// TIA Portal V15.1 export
// export: Created 2022-12-20T09:13:23.2931876Z, ExportSetting None, DisplayName Totally Integrated Automation Portal, DisplayVersion V15.1 Update 1, DisplayName TIA Portal Openness, DisplayVersion V15.1, DisplayName SINAMICS Startdrive Advanced, DisplayVersion V15.1, DisplayName G130, G150, S120, S150, SINAMICS MV, S210, DisplayVersion V15.1, DisplayName G110M, G120, G120C, G120D, G120P, DisplayVersion V15.1, DisplayName STEP 7 Professional, DisplayVersion V15.1 Update 1, DisplayName STEP 7 Safety, DisplayVersion V15.1, DisplayName WinCC Professional, DisplayVersion V15.1 Update 1, DisplayName SIMATIC Visualization Architect, DisplayVersion V15.1
FUNCTION_BLOCK "SA01_ESTOP_FB"   // FB901, FBD
TITLE = SA01_Estop_FB
{ S7_Optimized_Access := 'TRUE' }
// The block is used to control the estops that are located on SA01
// stored: AutoNumber false, MemoryReserve 100, SetENOAutomatically False
   VAR
      "xxx-xxxx" : "CM_Estop_FB";   // Emergency stop HMI load area xxxx
   END_VAR
BEGIN

REGION Network 1: Call emergency stop HMI load area Stxxx
   // E-stop xxxx
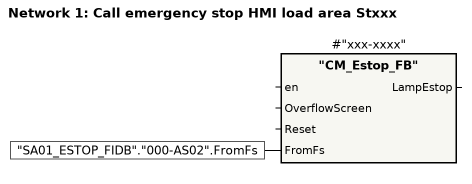
   #"xxx-xxxx"(FromFs := "SA01_ESTOP_FIDB"."000-AS02".FromFs);   // "CM_Estop_FB"
END_REGION
END_FUNCTION_BLOCK
